(* IEC 61131-3 sources: traffic-lights/PLC_TrafficLights/Class/TrafficLight, 1 file *)

(* ---- TrafficLight.st ---- *)
(*!
<Class
	Name               = "TrafficLight"
	Revision           = "0.0"
	RealtimeTask       = "false"
	CyclicTask         = "true"
	DefCyclictime      = "100 ms"
	BackgroundTask     = "false"
	Sigmatek           = "false"
	OSInterface        = "false"
	HighPriority       = "false"
	Automatic          = "false"
	UpdateMode         = "Prescan"
	SharedCommandTable = "true"
	Objectsize         = "(496,120)">
	<Channels>
		<Server Name="ClassSvr" Visualized="false" Initialize="false" WriteProtected="true" Retentive="false"/>
		<Server Name="Svr_Light" Visualized="true" Initialize="true" DefValue="0" WriteProtected="false" Retentive="false"/>
		<Server Name="Svr_SwitchDelay" Visualized="false" Initialize="true" DefValue="1500" WriteProtected="false" Retentive="SRam"/>
	</Channels>
</Class>
*)
TrafficLight : CLASS
	TYPE
	  _LightColor :  //! <Type Public="true" Name="_LightColor"/>
	  (
	    eRed:=0,
	    eYellow:=1,
	    eGreen:=2
	  )$DINT;
	END_TYPE
  //Servers:
	ClassSvr 	: SvrChCmd_DINT;
	Svr_Light 	: SvrCh__LightColor_PTofCls_TrafficLight;
	Svr_SwitchDelay 	: SvrCh_UDINT;
  //Clients:
  //Variables:
		tSignalChanged 	: UDINT;
		bStopSignal 	: BOOL;
  //Functions:

	FUNCTION VIRTUAL GLOBAL CyWork
		VAR_INPUT
			EAX 	: UDINT;
		END_VAR
		VAR_OUTPUT
			state (EAX) 	: UDINT;
		END_VAR;

	FUNCTION GLOBAL SetSignal
		VAR_INPUT
			ShouldStop 	: BOOL;
		END_VAR;
  //Tables:
	FUNCTION @STD
		VAR_OUTPUT
			ret_code	: CONFSTATES;
		END_VAR;
	FUNCTION GLOBAL TAB @CT_;
END_CLASS;

//----------------------------------------------------------------------------------------------------
//  Standard class methods
//----------------------------------------------------------------------------------------------------

// Standard Cywork, runs every set amount of time.
FUNCTION VIRTUAL GLOBAL TrafficLight::CyWork
	VAR_INPUT
		EAX 	: UDINT;
	END_VAR
	VAR_OUTPUT
		state (EAX) 	: UDINT;
	END_VAR

        CASE Svr_Light OF

        // Svr_Light is Green -> Yellow
        eGreen:
            IF bStopSignal THEN
                Svr_Light.Write(eYellow);
            END_IF;

        // Svr_Light is Yellow -> Red
        eYellow:
            IF (OPS.tAbsolute - tSignalChanged) > Svr_SwitchDelay THEN
                Svr_Light.Write(eRed);
            END_IF;

        // Svr_Light is Red -> Green
        eRed:
            IF bStopSignal = FALSE & (OPS.tAbsolute - tSignalChanged) > Svr_SwitchDelay THEN
                Svr_Light.Write(eGreen);
            END_IF;
        END_CASE;

	state := READY;

END_FUNCTION

//----------------------------------------------------------------------------------------------------
//  Externally called methods
//----------------------------------------------------------------------------------------------------

// Sets the signal so the traffic light can turn to the right color.
FUNCTION GLOBAL TrafficLight::SetSignal
	VAR_INPUT
		ShouldStop 	: BOOL;
	END_VAR

    IF bStopSignal = ShouldStop THEN
        RETURN;
    END_IF;

    bStopSignal := ShouldStop;
    tSignalChanged := OPS.tAbsolute;

END_FUNCTION
